// LS Electric XG5000 project: 64_1
// PLC NewPLC
// module base 0 slot 0: 입출력 모듈:XBC-DR14E (DC 24V 입력 8점, 릴레이 출력 6점)

PROGRAM NewProgram (task: 스캔 프로그램)

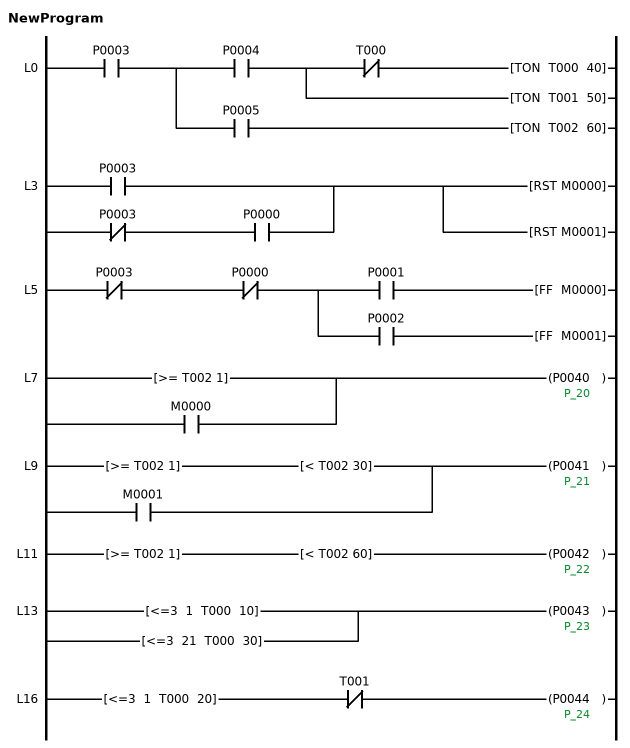
; L0
LOAD      P0003
MPUSH
AND       P0004
MPUSH
AND NOT   T000
TON       T000 40
MPOP
TON       T001 50
MPOP
AND       P0005
TON       T002 60
; L3
LOAD      P0003
LOAD NOT  P0003
AND       P0000
OR LOAD
RST       M0000
RST       M0001
; L5
LOAD NOT  P0003
AND NOT   P0000
MPUSH
AND       P0001
FF        M0000
MPOP
AND       P0002
FF        M0001
; L7
LOAD>=    T002 1
OR        M0000
OUT       P0040	// P_20
; L9
LOAD>=    T002 1
AND<      T002 30
OR        M0001
OUT       P0041	// P_21
; L11
LOAD>=    T002 1
AND<      T002 60
OUT       P0042	// P_22
; L13
LOAD<=3   1 T000 10
OR<=3     21 T000 30
OUT       P0043	// P_23
; L16
LOAD<=3   1 T000 20
AND NOT   T001
OUT       P0044	// P_24